PROGRAM MAIN
VAR
	enable AT%Q* : BOOL;
	speed AT%Q* : INT;
	motor_aan AT%Q* : INT;
END_VAR

motor();

ACTION motor:
speed := 20000;

IF enable = TRUE THEN
	motor_aan := speed;
END_IF;
END_ACTION

END_PROGRAM

(* stored: Version 1.1.0.1, ProductVersion 3.1.4024.9
   POU MAIN: Id {73d23b6c-8b30-4588-8b3a-0edb20e25878}, SpecialFunc None
   Action motor: Id {cc3ce1ad-8f58-4bd2-ad22-b2c7c999bb6b} *)
